TYPE ST_HMI :
STRUCT
	
	stMachine_Ctrl						:ST_MachineControl;
	stSP_Machine_Ctrl					:ST_MachineControl;
	stBatch_Ctrl						:ST_BatchControl;

	stReport_Ctrl						:ST_ReportControl;
	stProcess_Ctrl						:ST_ProcessControl;
	stAlarm_Ctrl						:ST_AlarmControl;
	
	iSelectedPhase						:INT;
	bCloseHMI							:BOOL;
	bScreenshot							:BOOL;
	bScanBatchParams					:BOOL;
	bReadCapacity						:BOOL;
		
END_STRUCT
END_TYPE

(* stored: Version 1.1.0.1, ProductVersion 3.1.4026.13
   DUT ST_HMI: Id {c99a5bf1-1e99-4d85-a667-5c2f839af9bd} *)
